# EPICS substitutions: sampleApp/Db/m1/2posActuator.substitutions
file vici_2pos_move.template {
    { DEV = $(DEV),PORT = $(PORT)}
}

file vici_settings.template {
    { DEV=$(DEV),PORT=$(PORT) }
}
#the scan sub will adjust how fast the current position readback is scanned
file vici_settings.template {
    {DEV=$(DEV),PORT=$(PORT), SCAN="1 second"  }
}
